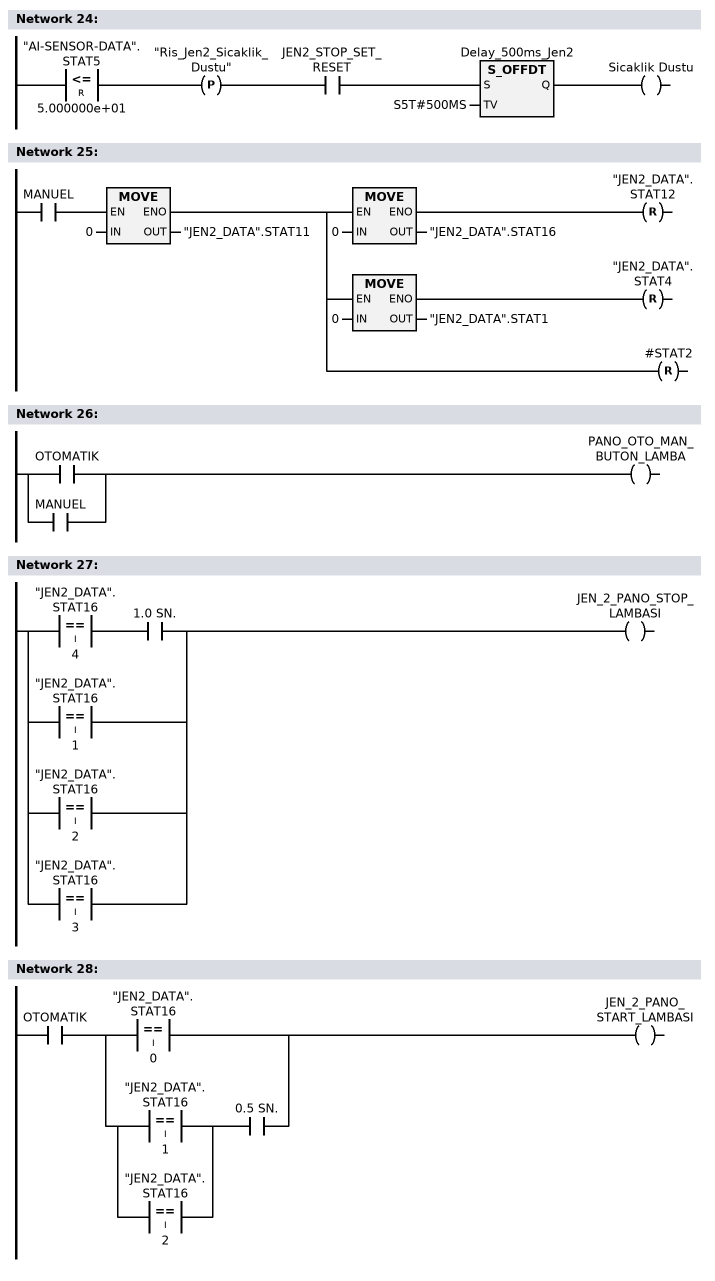
NETWORK
TITLE =
      A(;
      L     "AI-SENSOR-DATA".STAT5;
      L     5.000000e+01;
      <=R;
      );
      FP    "Ris_Jen2_Sicaklik_Dustu";
      A     "JEN2_STOP_SET_RESET";
      L     S5T#500MS;
      SF    "Delay_500ms_Jen2";
      NOP   0;
      NOP   0;
      NOP   0;
      A     "Delay_500ms_Jen2";
      =     "Sicaklik Dustu";
NETWORK
TITLE =
      A     "MANUEL";
      JNB   _018;
      L     0;
      T     "JEN2_DATA".STAT11;
      SET;
      SAVE;
      CLR;
_018: A     BR;
      =     L 0.0;
      A     L 0.0;
      JNB   _019;
      L     0;
      T     "JEN2_DATA".STAT16;
      SET;
      SAVE;
      CLR;
_019: A     BR;
      R     "JEN2_DATA".STAT12;
      A     L 0.0;
      JNB   _01a;
      L     0;
      T     "JEN2_DATA".STAT1;
      SET;
      SAVE;
      CLR;
_01a: A     BR;
      R     "JEN2_DATA".STAT4;
      A     L 0.0;
      BLD   102;
      R     #STAT2;
NETWORK
TITLE =
      O     "OTOMATIK";
      O     "MANUEL";
      =     "PANO_OTO_MAN_BUTON_LAMBA";
NETWORK
TITLE =
      A(;
      L     "JEN2_DATA".STAT16;
      L     4;
      ==I;
      );
      A     "1.0 SN.";
      O(;
      L     "JEN2_DATA".STAT16;
      L     1;
      ==I;
      );
      O(;
      L     "JEN2_DATA".STAT16;
      L     2;
      ==I;
      );
      O(;
      L     "JEN2_DATA".STAT16;
      L     3;
      ==I;
      );
      =     "JEN_2_PANO_STOP_LAMBASI";
NETWORK
TITLE =
      A     "OTOMATIK";
      A(;
      O(;
      L     "JEN2_DATA".STAT16;
      L     0;
      ==I;
      );
      O;
      A(;
      O(;
      L     "JEN2_DATA".STAT16;
      L     1;
      ==I;
      );
      O(;
      L     "JEN2_DATA".STAT16;
      L     2;
      ==I;
      );
      );
      A     "0.5 SN.";
      );
      =     "JEN_2_PANO_START_LAMBASI";
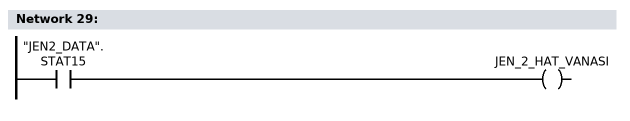
NETWORK
TITLE =
      A     "JEN2_DATA".STAT15;
      =     "JEN_2_HAT_VANASI";
END_FUNCTION_BLOCK

FUNCTION "TIME_UNSCALE" : VOID	// FC 1
VERSION : 0.0
BEGIN
// body was compiled from an SCL source; compiled code not shown
END_FUNCTION

FUNCTION "O.Vana_AciklikHesaplama" : VOID	// FC 2
VERSION : 0.1
VAR_INPUT
  IlkAciklikDegeri : REAL ;
  KademeliAcikDegeri : REAL ;
END_VAR
VAR_OUTPUT
  oKademe_1 : REAL ;
  oKademe_2 : REAL ;
  oKademe_3 : REAL ;
  oKademe_4 : REAL ;
  oKademe_5 : REAL ;
  oKademe_6 : REAL ;
  oKademe_7 : REAL ;
END_VAR
VAR_TEMP
  tKademe : STRUCT
   Iki : REAL ;
   Uc : REAL ;
   Dort : REAL ;
   Bes : REAL ;
   Alti : REAL ;
   Yedi : REAL ;
  END_STRUCT ;
  tCheck_Kademe5 : BOOL ;
  tCheck_Kademe6 : BOOL ;
  tCheck_Kademe7 : BOOL ;
END_VAR
BEGIN
NETWORK
TITLE =
//------------------------
// kademe 1
      L     #IlkAciklikDegeri;
      T     #oKademe_1;
//------------------------
// kademe 2
      L     #IlkAciklikDegeri;
      L     #KademeliAcikDegeri;
      +R;
      T     #tKademe.Iki;
      L     #tKademe.Iki;
      T     #oKademe_2;
//-----------------------
// kademe 3
      L     #KademeliAcikDegeri;
      L     #tKademe.Iki;
      +R;
      T     #tKademe.Uc;
      L     #tKademe.Uc;
      T     #oKademe_3;
//-----------------------
// kademe 4
      L     #KademeliAcikDegeri;
      L     #tKademe.Uc;
      +R;
      T     #tKademe.Dort;
      L     #tKademe.Dort;
      T     #oKademe_4;
//-----------------------
// kademe 5
      L     #KademeliAcikDegeri;
      L     #tKademe.Dort;
      +R;
      T     #tKademe.Bes;
      L     #tKademe.Bes;
      L     6.000000e+01;
      >R;
      =     #tCheck_Kademe5;
      A     #tCheck_Kademe5;
      JNB   j005;
      L     6.000000e+01;
      T     #tKademe.Bes;
j005: NOP   0;
      L     #tKademe.Bes;
      T     #oKademe_5;
//-----------------------
// kademe 6
      L     #KademeliAcikDegeri;
      L     #tKademe.Bes;
      +R;
      T     #tKademe.Alti;
      L     #tKademe.Alti;
      L     6.000000e+01;
      >R;
      =     #tCheck_Kademe6;
      A     #tCheck_Kademe6;
      JNB   j006;
      L     6.000000e+01;
      T     #tKademe.Alti;
j006: NOP   0;
      L     #tKademe.Alti;
      T     #oKademe_6;
//-----------------------
// kademe 7
      L     #KademeliAcikDegeri;
      L     #tKademe.Alti;
      +R;
      T     #tKademe.Yedi;
      L     #tKademe.Yedi;
      L     6.000000e+01;
      >R;
      =     #tCheck_Kademe7;
      A     #tCheck_Kademe7;
      JNB   j007;
      L     6.000000e+01;
      T     #tKademe.Yedi;
j007: NOP   0;
      L     #tKademe.Yedi;
      T     #oKademe_7;
NETWORK
TITLE =
END_FUNCTION

FUNCTION "Int_To_S5Time" : VOID	// FC 10
VERSION : 0.0
VAR_INPUT
  Saat : INT ;
  Dakika : INT ;
END_VAR
VAR_OUTPUT
  HesaplananSure_S5TIME : S5TIME ;
END_VAR
VAR_TEMP
  tSaat_Dint : DINT ;
  tHesaplananSaat : DINT ;
  tDakika_Dint : DINT ;
  tHesaplananDakika : DINT ;
  tHesaplnananSure_Dint : DINT ;
  tHesaplananSure_Time : TIME ;
END_VAR
BEGIN
// body was compiled from an SCL source; compiled code not shown
END_FUNCTION

// FC 33: know-how protected block, not included

// FC 40: know-how protected block, not included

// FC 105: know-how protected block, not included

// FC 106: know-how protected block, not included

DATA_BLOCK "AI-SENSOR-DATA"	// DB 1
VERSION : 0.1
  STRUCT
   STAT0 : REAL ;
   STAT1 : REAL ;
   STAT2 : WORD ;
   STAT3 : WORD ;
   STAT4 : REAL ;
   STAT5 : REAL ;
   STAT6 : WORD ;
   STAT7 : WORD ;
   STAT8 : REAL ;
   STAT9 : REAL ;
   STAT10 : WORD ;
   STAT11 : WORD ;
   STAT12 : WORD ;
   STAT13 : REAL ;
   STAT14 : WORD ;
   STAT15 : REAL ;
   STAT16 : BOOL ;
  END_STRUCT ;	
BEGIN
   STAT0 := 4.452402e+00;
   STAT3 := W#16#8;
   STAT4 := 1.514829e+02;
   STAT5 := 2.052228e+01;
   STAT8 := 5.423901e+01;
   STAT9 := 9.780092e+00;
   STAT13 := 4.622757e+00;
   STAT15 := 4.994936e+00;
   STAT16 := TRUE;
END_DATA_BLOCK

DATA_BLOCK "ORTAK_DATA"	// DB 2
VERSION : 0.1
  STRUCT
   STAT0 : REAL ;
   STAT1 : REAL ;
   STAT2 : REAL ;
   STAT3 : REAL ;
   STAT4 : BOOL ;
   STAT5 : REAL ;
  END_STRUCT ;	
BEGIN
END_DATA_BLOCK

DATA_BLOCK "TIME_OTO_1_DB"	// DB 5
AUTHOR : SIMATIC
FAMILY : IEC_TC
VERSION : 0.0
"TON"
BEGIN
END_DATA_BLOCK

DATA_BLOCK "TIME_OTO_2_DB"	// DB 6
AUTHOR : SIMATIC
FAMILY : IEC_TC
VERSION : 0.0
"TON"
BEGIN
END_DATA_BLOCK

DATA_BLOCK "TIME_OTO_1_PROSES_DB"	// DB 7
AUTHOR : SIMATIC
FAMILY : IEC_TC
VERSION : 0.0
"TON"
BEGIN
END_DATA_BLOCK

DATA_BLOCK "TIME_OTO_2_PROSES_DB"	// DB 8
AUTHOR : SIMATIC
FAMILY : IEC_TC
VERSION : 0.0
"TON"
BEGIN
END_DATA_BLOCK

DATA_BLOCK DB 9
AUTHOR : SIMATIC
FAMILY : IEC_TC
VERSION : 0.0
"TON"
BEGIN
END_DATA_BLOCK

DATA_BLOCK DB 10
AUTHOR : SIMATIC
FAMILY : IEC_TC
VERSION : 0.0
"TON"
BEGIN
END_DATA_BLOCK

DATA_BLOCK "SURELER_DB"	// DB 14
VERSION : 0.0
"SURELER"
BEGIN
END_DATA_BLOCK

DATA_BLOCK "SAFETY_DB"	// DB 15
VERSION : 0.0
"SAFETY"
BEGIN
END_DATA_BLOCK

DATA_BLOCK "KAZAN1_DATA"	// DB 17
VERSION : 0.1
  STRUCT
   STAT0 : INT ;
   STAT1 : BOOL ;
   STAT2 : BOOL ;
   STAT3 : S5TIME ;
   STAT4 : INT ;
   STAT5 : REAL ;
   STAT6 : REAL ;
   STAT7 : BOOL ;
   STAT8 : REAL ;
   STAT9 : BOOL ;
   STAT10 : WORD ;
   STAT11 : REAL ;
   STAT12 : BOOL ;
   STAT13 : WORD ;
   STAT14 : REAL ;
   STAT15 : INT ;
   STAT16 : BOOL ;
   STAT17 : BOOL ;
   STAT18 : BOOL ;
   STAT19 : BOOL ;
   STAT20 : TIME ;
   STAT21 : DINT ;
   STAT22 : TIME ;
   STAT23 : DINT ;
   STAT24 : TIME ;
   STAT25 : DINT ;
  END_STRUCT ;	
BEGIN
   STAT1 := TRUE;
   STAT3 := S5T#21M;
   STAT4 := 3;
   STAT5 := 4.500000e+00;
   STAT6 := 3.616898e-03;
   STAT11 := 3.978588e-03;
   STAT14 := 5.775463e+01;
   STAT15 := 7969;
   STAT21 := L#1260;
END_DATA_BLOCK

DATA_BLOCK "KAZAN2_DATA"	// DB 18
VERSION : 0.1
  STRUCT
   STAT0 : INT ;
   STAT1 : BOOL ;
   STAT2 : BOOL ;
   STAT3 : S5TIME ;
   STAT4 : INT ;
   STAT5 : REAL ;
   STAT6 : REAL ;
   STAT7 : BOOL ;
   STAT8 : REAL ;
   STAT9 : BOOL ;
   STAT10 : WORD ;
   STAT11 : REAL ;
   STAT12 : BOOL ;
   STAT13 : WORD ;
   STAT14 : REAL ;
   STAT15 : INT ;
   STAT16 : BOOL ;
   STAT17 : BOOL ;
   STAT18 : BOOL ;
   STAT19 : BOOL ;
   STAT20 : TIME ;
   STAT21 : DINT ;
   STAT22 : TIME ;
   STAT23 : DINT ;
   STAT24 : TIME ;
   STAT25 : DINT ;
  END_STRUCT ;	
BEGIN
   STAT1 := TRUE;
   STAT3 := S5T#21M;
   STAT4 := -23;
   STAT5 := 4.500000e+00;
   STAT6 := 2.857350e-02;
   STAT11 := 4.701968e-03;
   STAT14 := 1.045356e+02;
   STAT15 := 14476;
   STAT21 := L#1260;
END_DATA_BLOCK

DATA_BLOCK "JEN1_DATA"	// DB 19
VERSION : 0.1
  STRUCT
   STAT0 : REAL ;
   STAT1 : INT ;
   STAT2 : REAL ;
   STAT3 : REAL ;
   STAT4 : BOOL ;
   STAT5 : BOOL ;
   STAT6 : BOOL ;
   STAT7 : BOOL ;
   STAT8 : BOOL ;
   STAT9 : BOOL ;
   STAT10 : BOOL ;
   STAT11 : INT ;
   STAT12 : BOOL ;
   STAT13 : BOOL ;
   STAT14 : BOOL ;
   STAT15 : BOOL ;
   STAT16 : INT ;
   STAT17 : BOOL ;
   STAT18 : TIME ;
   STAT19 : DINT ;
   STAT20 : BOOL ;
   STAT21 : DINT ;
   STAT22 : BOOL ;
  END_STRUCT ;	
BEGIN
   STAT0 := 3.000000e+00;
   STAT2 := 1.050000e+02;
   STAT3 := 1.300000e+02;
   STAT11 := 1;
   STAT12 := TRUE;
   STAT13 := TRUE;
   STAT14 := TRUE;
   STAT15 := TRUE;
   STAT16 := 3;
   STAT19 := L#32124;
END_DATA_BLOCK

DATA_BLOCK "JEN2_DATA"	// DB 20
VERSION : 0.1
  STRUCT
   STAT0 : REAL ;
   STAT1 : INT ;
   STAT2 : REAL ;
   STAT3 : REAL ;
   STAT4 : BOOL ;
   STAT5 : BOOL ;
   STAT6 : BOOL ;
   STAT7 : BOOL ;
   STAT8 : BOOL ;
   STAT9 : BOOL ;
   STAT10 : BOOL ;
   STAT11 : INT ;
   STAT12 : BOOL ;
   STAT13 : BOOL ;
   STAT14 : BOOL ;
   STAT15 : BOOL ;
   STAT16 : INT ;
   STAT17 : BOOL ;
   STAT18 : TIME ;
   STAT19 : DINT ;
   STAT20 : BOOL ;
   STAT21 : DINT ;
  END_STRUCT ;	
BEGIN
   STAT0 := 3.000000e+00;
   STAT2 := 5.500000e+01;
   STAT3 := 1.100000e+02;
END_DATA_BLOCK

DATA_BLOCK "JEN1_PID_DATA"	// DB 21
VERSION : 0.1
  STRUCT
   STAT0 : REAL ;
   STAT1 : INT ;
  END_STRUCT ;	
BEGIN
END_DATA_BLOCK

DATA_BLOCK "JEN2_PID_DATA"	// DB 22
VERSION : 0.1
  STRUCT
   STAT0 : REAL ;
   STAT1 : INT ;
  END_STRUCT ;	
BEGIN
   STAT1 := 11059;
END_DATA_BLOCK

DATA_BLOCK "KAZAN1_PID_DATA"	// DB 23
VERSION : 0.1
  STRUCT
   STAT0 : INT ;
   STAT1 : REAL ;
  END_STRUCT ;	
BEGIN
END_DATA_BLOCK

DATA_BLOCK "KAZAN2_PID_DATA"	// DB 24
VERSION : 0.1
  STRUCT
   STAT0 : INT ;
   STAT1 : REAL ;
  END_STRUCT ;	
BEGIN
END_DATA_BLOCK

DATA_BLOCK DB 50
AUTHOR : SIMATIC
FAMILY : ICONT
VERSION : 0.0
"CONT_C"
BEGIN
END_DATA_BLOCK

DATA_BLOCK "JEN2_KONTROL_BLOGU_DB"	// DB 51
VERSION : 0.0
"JEN2_PID_KONTROL"
BEGIN
END_DATA_BLOCK

DATA_BLOCK DB 52
VERSION : 0.0
"JEN1_PID_KONTROL"
BEGIN
END_DATA_BLOCK

DATA_BLOCK "JEN_1_PID_DB"	// DB 69
AUTHOR : SIMATIC
FAMILY : CONTROL
VERSION : 0.0
"TCONT_CP"
BEGIN
END_DATA_BLOCK

DATA_BLOCK "JEN_2_PID_DB"	// DB 70
AUTHOR : SIMATIC
FAMILY : CONTROL
VERSION : 0.0
"TCONT_CP"
BEGIN
END_DATA_BLOCK

DATA_BLOCK "OTOKLAV_1_DB"	// DB 94
VERSION : 0.0
"KAZAN_1_KONTROL"
BEGIN
END_DATA_BLOCK

DATA_BLOCK "OTOKLAV_2_DB"	// DB 95
VERSION : 0.0
"KAZAN_2_KONTROL"
BEGIN
END_DATA_BLOCK

DATA_BLOCK "FB98_DB"	// DB 98
VERSION : 0.0
"JEN1_KONTROL_BLOGU"
BEGIN
END_DATA_BLOCK

DATA_BLOCK "FB99_DB"	// DB 99
VERSION : 0.0
"JEN2_KONTROL_BLOGU"
BEGIN
END_DATA_BLOCK

DATA_BLOCK "HMI_DATA"	// DB 100
VERSION : 0.1
  STRUCT
   JEN1_Min_Basinc : REAL  := 5.000000e+000;	//Jenerator 1 min otomatik sekans basinci
   JEN1_Max_Basinc : REAL  := 5.500000e+000;	//Jenerator 1 max otomatik sekans basinci
   JEN2_Min_Basinc : REAL  := 5.000000e+000;	//Jenerator 2 min otomatik sekans basinci
   JEN2_Max_Basinc : REAL  := 5.500000e+000;	//Jenerator 2 max otomatik sekans basinci
   OTOKLAV_First_Oran : REAL  := 2.000000e+001;	//Otoklav oransal vana otomatik sekans ilk acilis orani
   OTOKLAV_Kademeli_Artis : REAL  := 5.000000e+000;	//Otoklav oransal vana kademeli artis katsayisi
   Otoklav_1_TimeData : STRUCT 	//Otoklav 1 hmi süre bilgisi
    Hours : INT ;	//Istenen calisma saati
    Minutes : INT  := 30;	//Istenen calisma dakikasi
    Second : INT ;	//Istenen calisma saniyesi
   END_STRUCT ;
   Otoklav_2_TimeData : STRUCT 	//Otoklav 2 hmi süre bilgisi
    Hours : INT ;	//Istenen calisma saati
    Minutes : INT  := 30;	//Istenen calisma dakikasi
    Second : INT ;	//Istenen calisma saniyesi
   END_STRUCT ;
   O_VanaAciklikOrani : REAL  := 2.500000e+001;	//Oransal vana aciklik orani
   O_VanaKademeSayisi : REAL  := 5.000000e+000;	//Oransal vana kademeli artis katsayisi
  END_STRUCT ;	
BEGIN
   JEN1_Min_Basinc := 5.000000e+00;
   JEN1_Max_Basinc := 5.500000e+00;
   JEN2_Min_Basinc := 5.000000e+00;
   JEN2_Max_Basinc := 5.500000e+00;
   Otoklav_1_TimeData.Minutes := 30;
   Otoklav_2_TimeData.Minutes := 30;
END_DATA_BLOCK

DATA_BLOCK DB 120
VERSION : 0.0
"KAZAN_ORTAK"
BEGIN
END_DATA_BLOCK

DATA_BLOCK "KAZAN_1_PID_DB"	// DB 130
AUTHOR : SIMATIC
FAMILY : CONTROL
VERSION : 0.0
"TCONT_CP"
BEGIN
END_DATA_BLOCK

DATA_BLOCK DB 131
VERSION : 0.0
"KAZAN_1_PID_KONTROL"
BEGIN
END_DATA_BLOCK

DATA_BLOCK DB 132
VERSION : 0.0
"KAZAN_2_PID_KONTROL"
BEGIN
END_DATA_BLOCK

DATA_BLOCK DB 230
VERSION : 0.0
"KAZAN_ORTAK"
BEGIN
END_DATA_BLOCK

DATA_BLOCK "KAZAN_2_PID_DATA"	// DB 231
AUTHOR : SIMATIC
FAMILY : CONTROL
VERSION : 0.0
"TCONT_CP"
BEGIN
END_DATA_BLOCK

DATA_BLOCK DB 232
VERSION : 0.0
"TEST_BLOGU"
BEGIN
END_DATA_BLOCK

ORGANIZATION_BLOCK OB 1
VERSION : 0.1
VAR_TEMP
  TEMP0 : BYTE ;
  TEMP1 : BYTE ;
  TEMP2 : BYTE ;
  TEMP3 : BYTE ;
  TEMP4 : BYTE ;
  TEMP5 : BYTE ;
  TEMP6 : INT ;
  TEMP7 : INT ;
  TEMP8 : INT ;
  TEMP9 : DATE_AND_TIME ;
END_VAR
BEGIN
NETWORK
TITLE =
      UC    "MAINBLOCK";
NETWORK
TITLE =
      CALL  "SCALE" (
           $1                       := P#P 292.0,
           $2                       := L#1092616192,
           $3                       := L#0,
           $4                       := "ALWAYS OFF",
           $5                       := "AI-SENSOR-DATA".STAT12,
           $6                       := "AI-SENSOR-DATA".STAT13);
      CALL  "SCALE" (
           $1                       := P#P 294.0,
           $2                       := L#1092616192,
           $3                       := L#0,
           $4                       := "ALWAYS OFF",
           $5                       := "AI-SENSOR-DATA".STAT14,
           $6                       := "AI-SENSOR-DATA".STAT15);
NETWORK
TITLE =
END_ORGANIZATION_BLOCK

ORGANIZATION_BLOCK "PID BLOCK"	// OB 35
VERSION : 0.1
VAR_TEMP
  TEMP0 : BYTE ;
  TEMP1 : BYTE ;
  TEMP2 : BYTE ;
  TEMP3 : BYTE ;
  TEMP4 : BYTE ;
  TEMP5 : BYTE ;
  TEMP6 : WORD ;
  TEMP7 : INT ;
  TEMP8 : INT ;
  TEMP9 : DATE_AND_TIME ;
END_VAR
BEGIN
NETWORK
TITLE =
      CALL  "JEN1_PID_KONTROL" , DB 52;
      CALL  "JEN2_PID_KONTROL" , "JEN2_KONTROL_BLOGU_DB";
NETWORK
TITLE =
      CALL  "KAZAN_1_PID_KONTROL" , DB 131;
      CALL  "KAZAN_2_PID_KONTROL" , DB 132;
END_ORGANIZATION_BLOCK

ORGANIZATION_BLOCK "ZAMANHATASI"	// OB 80
VERSION : 0.1
VAR_TEMP
  TEMP0 : BYTE ;
  TEMP1 : BYTE ;
  TEMP2 : BYTE ;
  TEMP3 : BYTE ;
  TEMP4 : BYTE ;
  TEMP5 : BYTE ;
  TEMP6 : WORD ;
  TEMP7 : BYTE ;
  TEMP8 : BYTE ;
  TEMP9 : BYTE ;
  TEMP10 : BYTE ;
  TEMP11 : DATE_AND_TIME ;
END_VAR
BEGIN
NETWORK
TITLE =
END_ORGANIZATION_BLOCK

ORGANIZATION_BLOCK "GERILIMHATASI"	// OB 81
VERSION : 0.1
VAR_TEMP
  TEMP0 : BYTE ;
  TEMP1 : BYTE ;
  TEMP2 : BYTE ;
  TEMP3 : BYTE ;
  TEMP4 : BYTE ;
  TEMP5 : BYTE ;
  TEMP6 : WORD ;
  TEMP7 : BYTE ;
  TEMP8 : BYTE ;
  TEMP9 : BYTE ;
  TEMP10 : BYTE ;
  TEMP11 : DATE_AND_TIME ;
END_VAR
BEGIN
NETWORK
TITLE =
END_ORGANIZATION_BLOCK

ORGANIZATION_BLOCK "HATAUYARISI"	// OB 82
VERSION : 0.1
VAR_TEMP
  TEMP0 : BYTE ;
  TEMP1 : BYTE ;
  TEMP2 : BYTE ;
  TEMP3 : BYTE ;
  TEMP4 : BYTE ;
  TEMP5 : BYTE ;
  TEMP6 : WORD ;
  TEMP7 : BOOL ;
  TEMP8 : BOOL ;
  TEMP9 : BOOL ;
  TEMP10 : BOOL ;
  TEMP11 : BOOL ;
  TEMP12 : BOOL ;
  TEMP13 : BOOL ;
  TEMP14 : BOOL ;
  TEMP15 : BYTE ;
  TEMP16 : BOOL ;
  TEMP17 : BOOL ;
  TEMP18 : BOOL ;
  TEMP19 : BOOL ;
  TEMP20 : BOOL ;
  TEMP21 : BOOL ;
  TEMP22 : BOOL ;
  TEMP23 : BOOL ;
  TEMP24 : BOOL ;
  TEMP25 : BOOL ;
  TEMP26 : BOOL ;
  TEMP27 : BOOL ;
  TEMP28 : BOOL ;
  TEMP29 : BOOL ;
  TEMP30 : BOOL ;
  TEMP31 : BOOL ;
  TEMP32 : DATE_AND_TIME ;
END_VAR
BEGIN
NETWORK
TITLE =
END_ORGANIZATION_BLOCK

ORGANIZATION_BLOCK "TAKMACIKARMAHATASI"	// OB 83
VERSION : 0.1
VAR_TEMP
  TEMP0 : BYTE ;
  TEMP1 : BYTE ;
  TEMP2 : BYTE ;
  TEMP3 : BYTE ;
  TEMP4 : BYTE ;
  TEMP5 : BYTE ;
  TEMP6 : WORD ;
  TEMP7 : INT ;
  TEMP8 : WORD ;
  TEMP9 : DATE_AND_TIME ;
END_VAR
BEGIN
NETWORK
TITLE =
END_ORGANIZATION_BLOCK

ORGANIZATION_BLOCK "CPUHARDWAREERROR"	// OB 84
VERSION : 0.1
VAR_TEMP
  TEMP0 : BYTE ;
  TEMP1 : BYTE ;
  TEMP2 : BYTE ;
  TEMP3 : BYTE ;
  TEMP4 : BYTE ;
  TEMP5 : BYTE ;
  TEMP6 : WORD ;
  TEMP7 : DWORD ;
  TEMP8 : DATE_AND_TIME ;
END_VAR
BEGIN
NETWORK
TITLE =
END_ORGANIZATION_BLOCK

ORGANIZATION_BLOCK "PROGRAMHATASI"	// OB 85
VERSION : 0.1
VAR_TEMP
  TEMP0 : BYTE ;
  TEMP1 : BYTE ;
  TEMP2 : BYTE ;
  TEMP3 : BYTE ;
  TEMP4 : BYTE ;
  TEMP5 : BYTE ;
  TEMP6 : INT ;
  TEMP7 : BYTE ;
  TEMP8 : BYTE ;
  TEMP9 : BYTE ;
  TEMP10 : BYTE ;
  TEMP11 : DATE_AND_TIME ;
END_VAR
BEGIN
NETWORK
TITLE =
END_ORGANIZATION_BLOCK

ORGANIZATION_BLOCK "RACKHATASI"	// OB 86
VERSION : 0.1
VAR_TEMP
  TEMP0 : BYTE ;
  TEMP1 : BYTE ;
  TEMP2 : BYTE ;
  TEMP3 : BYTE ;
  TEMP4 : BYTE ;
  TEMP5 : BYTE ;
  TEMP6 : WORD ;
  TEMP7 : ARRAY  [0 .. 31 ] OF BOOL ;
  TEMP8 : DATE_AND_TIME ;
END_VAR
BEGIN
NETWORK
TITLE =
END_ORGANIZATION_BLOCK

ORGANIZATION_BLOCK "HABERLESMEHATASI"	// OB 87
VERSION : 0.1
VAR_TEMP
  TEMP0 : BYTE ;
  TEMP1 : BYTE ;
  TEMP2 : BYTE ;
  TEMP3 : BYTE ;
  TEMP4 : BYTE ;
  TEMP5 : BYTE ;
  TEMP6 : WORD ;
  TEMP7 : DWORD ;
  TEMP8 : DATE_AND_TIME ;
END_VAR
BEGIN
NETWORK
TITLE =
END_ORGANIZATION_BLOCK

ORGANIZATION_BLOCK "COMPLETE RESTART"	// OB 100
VERSION : 0.1
VAR_TEMP
  TEMP0 : BYTE ;
  TEMP1 : BYTE ;
  TEMP2 : BYTE ;
  TEMP3 : BYTE ;
  TEMP4 : BYTE ;
  TEMP5 : BYTE ;
  TEMP6 : WORD ;
  TEMP7 : DWORD ;
  TEMP8 : DATE_AND_TIME ;
END_VAR
BEGIN
NETWORK
TITLE =
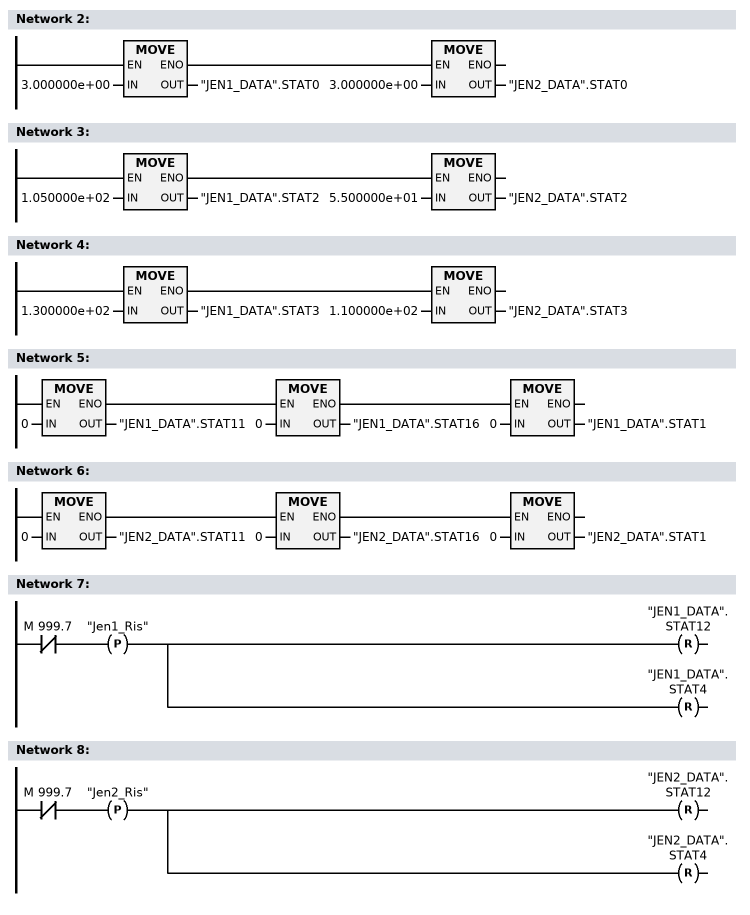
NETWORK
TITLE =
      A(;
      L     3.000000e+00;
      T     "JEN1_DATA".STAT0;
      SET;
      SAVE;
      CLR;
      A     BR;
      );
      JNB   _001;
      L     3.000000e+00;
      T     "JEN2_DATA".STAT0;
_001: NOP   0;
NETWORK
TITLE =
      A(;
      L     1.050000e+02;
      T     "JEN1_DATA".STAT2;
      SET;
      SAVE;
      CLR;
      A     BR;
      );
      JNB   _002;
      L     5.500000e+01;
      T     "JEN2_DATA".STAT2;
_002: NOP   0;
NETWORK
TITLE =
      A(;
      L     1.300000e+02;
      T     "JEN1_DATA".STAT3;
      SET;
      SAVE;
      CLR;
      A     BR;
      );
      JNB   _003;
      L     1.100000e+02;
      T     "JEN2_DATA".STAT3;
_003: NOP   0;
NETWORK
TITLE =
      A(;
      A(;
      L     0;
      T     "JEN1_DATA".STAT11;
      SET;
      SAVE;
      CLR;
      A     BR;
      );
      JNB   _004;
      L     0;
      T     "JEN1_DATA".STAT16;
      SET;
      SAVE;
      CLR;
_004: A     BR;
      );
      JNB   _005;
      L     0;
      T     "JEN1_DATA".STAT1;
_005: NOP   0;
NETWORK
TITLE =
      A(;
      A(;
      L     0;
      T     "JEN2_DATA".STAT11;
      SET;
      SAVE;
      CLR;
      A     BR;
      );
      JNB   _006;
      L     0;
      T     "JEN2_DATA".STAT16;
      SET;
      SAVE;
      CLR;
_006: A     BR;
      );
      JNB   _007;
      L     0;
      T     "JEN2_DATA".STAT1;
_007: NOP   0;
NETWORK
TITLE =
      AN    M 999.7;
      FP    "Jen1_Ris";
      R     "JEN1_DATA".STAT12;
      R     "JEN1_DATA".STAT4;
NETWORK
TITLE =
      AN    M 999.7;
      FP    "Jen2_Ris";
      R     "JEN2_DATA".STAT12;
      R     "JEN2_DATA".STAT4;
END_ORGANIZATION_BLOCK

ORGANIZATION_BLOCK "RESTART"	// OB 101
VERSION : 0.1
VAR_TEMP
  TEMP0 : BYTE ;
  TEMP1 : BYTE ;
  TEMP2 : BYTE ;
  TEMP3 : BYTE ;
  TEMP4 : BYTE ;
  TEMP5 : BYTE ;
  TEMP6 : WORD ;
  TEMP7 : DWORD ;
  TEMP8 : DATE_AND_TIME ;
END_VAR
BEGIN
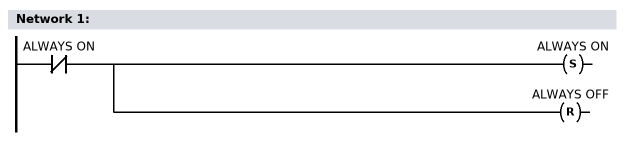
NETWORK
TITLE =
      AN    "ALWAYS ON";
      S     "ALWAYS ON";
      R     "ALWAYS OFF";
END_ORGANIZATION_BLOCK

ORGANIZATION_BLOCK "COLD RESTART"	// OB 102
VERSION : 0.1
VAR_TEMP
  TEMP0 : BYTE ;
  TEMP1 : BYTE ;
  TEMP2 : BYTE ;
  TEMP3 : BYTE ;
  TEMP4 : BYTE ;
  TEMP5 : BYTE ;
  TEMP6 : WORD ;
  TEMP7 : DWORD ;
  TEMP8 : DATE_AND_TIME ;
END_VAR
BEGIN
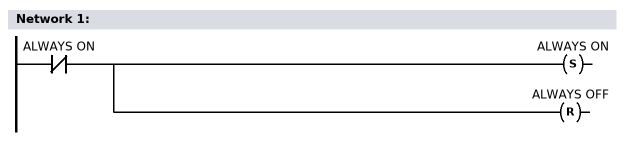
NETWORK
TITLE =
      AN    "ALWAYS ON";
      S     "ALWAYS ON";
      R     "ALWAYS OFF";
END_ORGANIZATION_BLOCK

ORGANIZATION_BLOCK "PROGRAMMINGERROR"	// OB 121
VERSION : 0.1
VAR_TEMP
  TEMP0 : BYTE ;
  TEMP1 : BYTE ;
  TEMP2 : BYTE ;
  TEMP3 : BYTE ;
  TEMP4 : BYTE ;
  TEMP5 : BYTE ;
  TEMP6 : WORD ;
  TEMP7 : WORD ;
  TEMP8 : WORD ;
  TEMP9 : DATE_AND_TIME ;
END_VAR
BEGIN
NETWORK
TITLE =
END_ORGANIZATION_BLOCK
